Staubli VAL3: JointFeedback.dtx

public num nRobotId
public num nValidFields
public num nTime
public num nPositions[10]
public num nVelocities[10]
public num nAccelerations[10]
